Staubli VAL3: listSetSize.pgx

public program listSetSize(num x_nPx, num x_nPy, num x_nPBottomX, num x_nPBottomY)
begin
  //-----------------------------------------------------------------------
  //Header begin
  //Description of program
  //  Defines all the parameters of positions and size of the list menu.
  //
  //Input parameters
  //  num x_nPx:
  //    role : cursor column position : top left corner for the beginning of
  //    the list menu
  //  num x_nPy :
  //    role : cursor column position : top left corner for the beginning of
  //    the list menu
  //  num x_nPBottomX
  //    role : width of the box
  //  num x_nPBottomY :
  //    role : height of the box
  //
  //Example
  //  call setSizeList(20,0,18,11)
  //
  //History
  //  Creation : 28-04-08 - f.Rob
  //Header end
  //-----------------------------------------------------------------------
  //Put all the parameters in globals variables
  nTopX=nTopX[1]=x_nPx
  nTopY=x_nPy
  nBottomX=nBottomX[1]=x_nPBottomX
  nListHeight=x_nPBottomY
end
